FUNCTION_BLOCK Plant
  (* Standard: 61499-2 *)
  (* Version 0.1, 2017-00-02, hpea485, UOA *)
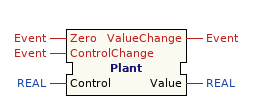
  EVENT_INPUT
    Zero;
    ControlChange;
  END_EVENT
  EVENT_OUTPUT
    ValueChange;
  END_EVENT
  VAR_INPUT
    Control : REAL;
  END_VAR
  VAR_OUTPUT
    Value : REAL;
  END_VAR
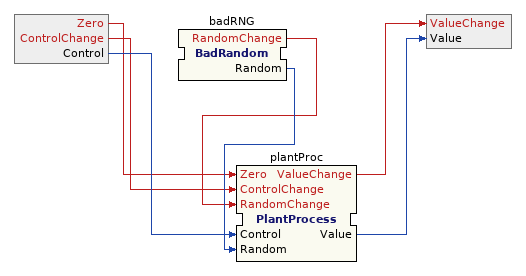
  FBS
    badRNG : BadRandom;
    plantProc : PlantProcess;
  END_FBS
  EVENT_CONNECTIONS
    Zero TO plantProc.Zero;
    ControlChange TO plantProc.ControlChange;
    plantProc.ValueChange TO ValueChange;
    badRNG.RandomChange TO plantProc.RandomChange;
  END_CONNECTIONS
  DATA_CONNECTIONS
    Control TO plantProc.Control;
    plantProc.Value TO Value;
    badRNG.Random TO plantProc.Random;
  END_CONNECTIONS
END_FUNCTION_BLOCK
